(* IEC 61131-3 sources: NachHouse_CORE/V200/APP (part 15) *)

				yBtn15 := xBtn15^;

							IF j > 7 THEN
								xR^.o.ob[j].y := xR^.o.ob[7].y;			// preberie suradnicu z objektu sviatok
							ELSIF j = 7 THEN
								xR^.o.ob[j].y := xR^.o.ob[0].y - 75;			// preberie suradnicu z objektu sviatok
							ELSIF j > 0 THEN
								xR^.o.ob[j].y := xR^.o.ob[0].y;        // preberie z Pondelok
							END_IF;
							IF xO^.fn > 0 THEN								// obrazky sviatok..dovolenka
								pp	:= xR^.o.ob[j].cf.n;;                	// cislo textu
  		            	   _NhVal2(obr	:= xO^.fn + BOOL_TO_INT(xPtB^),
  		               			wO		:= xO^.w,
                              grd   := 1,
                              box   := xPtB^,                   // kruh/kruznica
                              fil   := xPtB^,                	// bude vypln
                              BgC   := xO^.FgC,						// kruznica
                              FgC   := xO^.FgC,               	// vypln
//										wL		:= 2,                      // hrubka kruznice
//									   wC    := xO^.w*20/18,              		// wl=priemer gulicky, wl=hrubka kruznice
										hB    := xO^.w*20/18,
										r		:= 10,
											);
							ELSE                                 		// dni v tyzdni, nemaju vo .fn nic
								pp	:= 201;                					// textu: den v tyzdni
  		               	_NhVal2(
                              grd   := 2,
                              crc   := true,                   // kruh/kruznica
                              fil   := xPtB^,                	// bude vypln
                              BgC   := xO^.FgC,						// kruznica
                              FgC   := xO^.FgC,               	// vypln
										wL		:= 2,                      // hrubka kruznice
									   wC    := xO^.w,              		// wl=priemer gulicky, wl=hrubka kruznice

                              txt 	:= -2,
										nTxt 	:= 21 + SINT_TO_INT(j),	// 21=PO,UT,ST
										fmt   := 2,
                              FgT   := xO^.BgC,						// farba textu
                              wT    := xO^.w/2 );
							END_IF;
							IF xR^.o.ob[0].cf.c = 1 THEN 									// vykresli objekty kopirovania
				            GC_Move  (x := 24, y := -28, GrData := xCan);
					         IF xM^.pod.cp.src = i OR (xM^.pod.cp.all AND xM^.pod.cp.dst[i]) THEN				//
					            GC_CImage   (filename := _NhFnObr(fn := 44), width := 48, height := 48,	GrData := xCan);
								ELSIF xM^.pod.cp.src = 0 THEN
									;
					         ELSIF xM^.pod.cp.dst[i] THEN
				   	         GC_CImage   (filename := _NhFnObr(fn := 38), width := 45, height := 45,	GrData := xCan);
									xM^.pod.cp.cpy := true;									// centralny prinak, ze mame nejaky ciel
								END_IF;
								IF xM^.pod.cp.all = false AND xM^.pod.cp.cpy = false THEN
									xB^.r[1].o.ob[0].wh	:= 0;
								ELSE	 //xB^.r[1].o.ob[0].cm = 130 THEN					// menu kopirovania
									xB^.r[1].o.ob[0].wh	:= 1;
									IF xM^.pod.cp.all THEN
										xB^.r[1].o.ob[0].fn := 38;						// zeleny check
										xB^.r[1].o.ob[0].cm := 132;					// browser
									ELSE
										xB^.r[1].o.ob[0].fn := 44;              	// zlte copy
										xB^.r[1].o.ob[0].cm := 130;					// copy
									END_IF;
									xB^.r[1].o.ob[0].x	:= xR^.o.ob[6].x;       // preberie znedele
									xB^.r[1].o.ob[0].y	:=	xR^.o.ob[7].y-20;			// preberie suradnicu z objektu sviatok
					         END_IF;
							END_IF;

							IF pp > 0 AND xPtB^ AND xR^.o.ob[0].set6 THEN		// vypisuje sa text dna
  		               	_NhVal2(
										xy		:= true,
										x		:= xc,
										y		:= xR^.o.ob[7].y - xR^.o.ob[7].h,
                              txt 	:= -2,
										nTxt 	:= pp,
										fmt   := 2,
                              FgT   := 3,						// farba textu
                              wT    := 28 );
							END_IF;

      				END_IF;

           106:   // ikona typ.dna na Home/zone
                  xPtD  := ADR(xO^.cf.n); 	      // adresa premennej USINT;
						xPod	:= UDINT_TO_PTR(xPtD^);
						IF xPod^.Day < 8 THEN
	               	_NhVal2(wO:=xO^.w, obr:=269);					// cisty kalendar
	               	_NhVal2(
               			y		:= xO^.w/10,
                 			txt 	:= -2,
								nTxt 	:= 21 + USINT_TO_INT(xPod^.Day-1),
                        FgT   := 3,						// farba textu
								fmt   := 2,
                        wT   := xO^.w*10/26 );
						ELSE
	               	_NhVal2(
               			wO		:= xO^.w,
               			obr	:= 275 + (3*USINT_TO_INT(xPod^.Day-8)) );
						END_IF;

           221:  // Vypist textu s hodnotou
                  // xO^.fn      :  cislo textu vypisovane od pevne od x=50
						// ak xO^.cf.c > 0
	                  // xO^.cf.c    :  cfg DEV
   	               // xO^.cf.n    :  nd DEV
                  // xO^.FgC     :  farba textu
                  // xO^.w       :  vyska textu

                  // xO^.fmt     :  textova hodnota
                  // xO^.BgC     :  farba hodnoty
                  // xO^.h       :  vyska hodnoty

                  // xO^.x       :  x-obrazka
                  // xO^.y       :  y-textu aj obrazka

                  // xO^.BgC     :  x-ova suradnica zaciatku textu

                  yTx1 := '';
                  IF xO^.fn > 0 THEN
                     _Nh_Lang(id :=  xO^.fn ,txt := ADR(yTx1));
                  ELSIF xO^.cf.c > 0 THEN
                     IF _NhxPt(c:=xO^.cf.c, n:=xO^.cf.n, x:=81) THEN
                        aTrim(wht:=1,txt:=ADR(yTx1));
                        yTx1 := CONCAT(yTx1,' ',xPt^.cf.Name);
                        yTx1 := LEFT(yTx1,25);
                     END_IF;
                  END_IF;
                  IF yTx1 <> '' THEN
                     _NhVal2(txt:=0, fmt := 0, wt:= xO^.w, FgT := xO^.FgC ,xy:=true, x:=50, y:=xO^.y );
                  END_IF;
                  yTx1 := xO^.fmt;                                          // naformatuje hodnotu do textu
                  _NhVal2(txt:=0, fmt := 2, wt:= xO^.h, FgT := xO^.BgC, xy:=true, x:=x2-90, y:=xO^.y  );

           228:   // status [2] DEV v BRW,,Quick.... vsade
		            _Nh_FRM_Read(frm:=229);                        // obrazky pre typ NH_OBR_OPV
                  xHet  := xDev;
						CASE xR^.h.cf.c OF
                    6 : c:=0;
                  ELSE  c:=1;
                  END_CASE;
						o 		:= aCfg[xR^.h.cf.c].par;
						IF xR^.h.chk   THEN													// z webu nad regulatorm sa podhodi default par
							p := xR^.h.cf.p;
						ELSIF xO^.tch  THEN
							xDev^.al.in.par := xHet^.cf.par ;
							xDev^.al.ou.par := xHet^.cf.par ;
							p	:= xDev^.al.ou.par;
						ELSE
							p	:= xDev^.al.ou.par;
						END_IF;
						IF xO^.tch THEN
							xDev^.al.in.cmd := 1;
						END_IF;
						_NhxPar (cp := o , np := p,x:=-1006);
                  pHet  	:= xPar;
                  xPvA  	:= ADR(pHet^.par.pva);
						_NH_Het_Map_Reg();
                  _Nh_Shw_ini();
                  IF xDev^.cf.typ > _Nh_TYP THEN
                     xO^.fn      := 24;
                  ELSE
                     xO^.fn      := yFrm_229.reg[c].obr1[ xReg^.Mode, xRegMod^.wht, MIN(xDev^.al.sta,3)];
                  END_IF;
                  yRn.v[0].wO    := xO^.w;
                  yRn.v[0].obr   := xO^.fn;
                  yRn.v[0].wh    := 0;
                  _Nh_Shw_Val();

           230:   // hlavny obrazok DEV podla typu.  browse
                  yRn.v[0].wO    := xO^.w;
//						xO^.fn			:=_NhObrNbr(cf:=xO^.cf.c, t:=xDev^.cf.typ);
//							_NhTypObr(cf:=xO^.cf.c, typ:=xDev^.cf.typ);
//							xO^.fn := xObrWht^.obr;

                  _Nh_Shw_ini();

//                  yRn.v[0].obr   := xO^.fn;
//                  yRn.v[0].wh 	:= INT_TO_USINT(_NhObrNbr(cf:=xO^.cf.c, t:=xDev^.cf.typ, wh:=1));

						_NhTypObr(cf:=xO^.cf.c, typ:=xDev^.cf.typ);
						xO^.fn			:= xObrWht^.obr;
	               yRn.v[0].obr   := xObrWht^.obr;
                  yRn.v[0].wh 	:= xObrWht^.wht;

						IF yRn.v[0].wh > 0 THEN
							yRn.v[0].wO := xO^.w * 20 / 24;
//							yRn.v[0].wC := xO^.w * 20 / 20;
						ELSE
	                  yRn.v[0].wO := xO^.w;
						END_IF;

                  _Nh_Shw_Val();

           231:   // status [2] DEV v BRW,,Quick.... vsade

                  _Nh_FRM_Read(frm:=231);                      // funkcia naciatania do obr, ale strukturu 230
                  _Nh_Shw_ini();
						vr				:= xDev^.al.ou.val;
						vr		:= xDev^.al.OU.val;
						IF xR^.h.chk  AND aCfg[xR^.h.cf.c].ou THEN
							{$IFDEF __NH_DALI}
							IF xR^.h.cf.c = 43 AND xF^.cf.c = 44 THEN
			      	      dlgr  := _Nh_DL_sha(gr:=1, nd := xF^.cf.n)-100;                    // cislo GRP - 100
								xDLs 	:= xDEv;
								vr 	:= USINT_TO_REAL(xDLs^.cx.scn.lvl[dlgr]);
							ELSIF xR^.h.cf.c = 44 AND xF^.cf.c = 43 THEN
								dlgr  := _Nh_DL_sha(gr:=1, nd := xR^.h.cf.n)-100;                    // cislo GRP - 100
								_NhxPt(c:=xF^.cf.c, n:=xF^.cf.n,x:=-135);
								xDLs 	:= xPt;
								vr 	:= USINT_TO_REAL(xDLs^.cx.scn.lvl[dlgr]);
							ELSIF aCfg[xO^.cf.c].par > 0 THEN
							{$ELSE}
							IF aCfg[xO^.cf.c].par > 0 THEN
							{$END_IF}

                   		IF _NhxPar(cp := aCfg[xO^.cf.c].par, np := xR^.h.cf.p ,x:=238) THEN
									vr		:= USINT_TO_REAL(xPar^.all.lvl);
								ELSE
									;
//									vr		:= xDev^.al.ou.val);
								END_IF;
							END_IF;
							IF vr > 0.0  THEN
								yRn.v[0].txt 	:= 3;													// vypise sa to co je vo vr
								yRn.v[0].wh    := 21;												// pri check, je vzdy zeleny podklad
							ELSE
								yRn.v[0].wh  := 10;													// sivy podklad OFF
							END_IF;
						ELSE
	      				s 				:= xDev^.al.sta;
							IF s > 0 THEN
								s	:= 2;
							ELSE
								s	:= 0;
							END_IF;
							IF  yFrm_231.dev[xO^.cf.c,s] < 0 THEN
								p := yFrm_231.dev[xO^.cf.c,2] * -1  + USINT_TO_INT(xDev^.al.sta-1);
								p	:= MIN(p,50);						// opravit
								IF yFrm_231.sta[p, 0] < 0 THEN
		      	            yRn.v[0].txt   := INT_TO_SINT( yFrm_231.sta[p, 0] * -1 );
		         	         yRn.v[0].obr   := 0;
								ELSE
		               	   yRn.v[0].obr   := yFrm_231.sta[p, 0];
								END_IF;
  			               yRn.v[0].wh    := INT_TO_USINT(yFrm_231.sta[p, 1]);
(*
							ELSIF xO^.cf.c = 4 	AND vr < 100.0 THEN						// SCN nie je naplno
	         	         yRn.v[0].obr   := 0;
								IF vr  > 0.0 THEN
			         	      yRn.v[0].wh    := 11;
								ELSE
			         	      yRn.v[0].wh    := 10;
								END_IF;
*)
							ELSIF xO^.cf.c = 4  THEN						// SCN nie je naplno
								yRn.v[0].obr   := 207;
								IF vr >= 100.0 THEN
			         	      yRn.v[0].wh    := 14;
								ELSIF vr  > 0.0 THEN
			         	      yRn.v[0].wh    := 17;
								ELSE
									yRn.v[0].obr   := 0;
									yRn.v[0].wh    := 10;
								END_IF;

							ELSIF xO^.cf.c = 44 	AND vr < 100.0 THEN            			// DLg scen nie je naplno
	         	         yRn.v[0].obr   := 0;
								IF vr  > 0.0 THEN
			         	      yRn.v[0].wh    := 11;
								ELSE
			         	      yRn.v[0].wh    := 10;
								END_IF;
							ELSE
	         	         yRn.v[0].obr   := yFrm_231.dev[xO^.cf.c,s];
   	         	      yRn.v[0].wh    := INT_TO_USINT(yFrm_231.dev[xO^.cf.c,s+1]);
							END_IF;
						END_IF;

(*
						IF xO^.cf.c = 44 THEN														// DLg nema Check
							IF xDev^.al.ou.val >=254 THEN
								yRn.v[0].wh  := 102;													// Oranzovy ON = kompletne zapnuta scena
							END_IF;
                  ELSIF aCfg[xO^.cf.c].ou AND xR^.h.chk AND aCfg[xO^.cf.c].par > 0  THEN   // pre OUT-DEV vp vazbe
     						yRn.v[0].obr	:= 0;                                     // zrusi obrazok, aby sa nezmensoval podklad
							yRn.v[0].FgT   := 1;													// pri check, je vzdy zeleny podklad
							IF xF^.cf.c = 44 THEN
								yRn.v[0].wh    := 13;												// pri check, je vzdy zeleny podklad
								{$IFDEF __NH_DALI}
	 							dlgr	:= _Nh_DL_sha(gr:=1,nd := xF^.cf.n)-100 ;				// 0..15
								xDLg	:= xDev;
								vr		:= MIN(100,USINT_TO_REAL(xDLs^.cx.scn.LVL[ dlgr ]));
								IF vr > 0.0 THEN
									yRn.v[0].txt := 3;													// vypise sa to co je vo vr
								ELSE
									yRn.v[0].wh  := 10;													// sivy podklad OFF
								END_IF;
								{$END_IF}

                     ELSIF _NhxPar(cp := aCfg[xO^.cf.c].par, np := xR^.h.cf.p ,x:=238) THEN
								yRn.v[0].wh    := 13;												// pri check, je vzdy zeleny podklad
								vr	:= MIN(100,USINT_TO_REAL(xPar^.all.lvl));
								IF aCfg[xO^.cf.c].analog THEN
									yRn.v[0].txt := 3;													// vypise sa to co je vo vr
								ELSIF vr > 0.0 THEN
									yRn.v[0].txt := 2;													// vypise sa to co je vo vr
								ELSE
									yRn.v[0].wh  := 10;													// sivy podklad OFF
								END_IF
							END_IF;
                  END_IF;
*)
					   IF yRn.v[0].wh > 0 AND yRn.v[0].obr > 0 THEN								// obrazok ma podklad, zmensi sa
	                  yRn.v[0].wO := xO^.w*20/23;
					   END_IF;

                  _Nh_Shw_Val();

           232:   // HOME-DASH, Cat/hlavny obr + CAT/status
                  _Nh_FRM_Read(frm:=232);                      // funkcia naciatania do obr, ale strukturu 230
                  p := xO^.cf.n;                                                      // cislo CAT
						_NhxRoW(nbr := xA^.sbj, zon := true);
						_NhxZon(c:=3, nz:=xA^.sbj, x:=111);
						IF xRoW^.cat[p] THEN																// hlavna ikona   je j=1
							c := 1;
						ELSE
							c := 0;
						END_IF;

					   CASE p OF
                    6 : // PSN
								c := xZon^.cx.lck.stat;
								IF xZon^.cx.lck.stat > 9 THEN
									c := 2;
								ELSIF c = 2 AND xZon^.cx.lck.AllLocked = false THEN
									c := 10;
								END_IF;
		                  IF xL^.obj = 0 THEN
    								x4o   := ADR(xB^.r[4].o.ob[p]);
									x4o^	:= yFrm_232.psn4;
									ok		:= 0;
									IF xHoW^.BodyOu THEN
										x4o^.ok[1]  := 1;
										ok				:= 0;
									END_IF;
									IF xHoW^.BodyIn THEN
										x4o^.ok[2]  := 1;
										ok				:= 0;
									END_IF;
									_Nh_Shw_LCK_ET(sta:=xZon^.cx.lck.stat, et:=xZon^.cx.lck.et, o := 4);
									IF ok THEN
//										x4o^.wh	:= 0;
									END_IF
								END_IF;

                  ELSE
                  ;
                  END_CASE;
				  		_Nh_Shw_ini();
						_Nh_Shw_232(o1 := xL^.obj > 0 AND j=1,  cat := p, sta := c);     	// pre j=1 hlavna ikona sa je iny obrazok
                  _Nh_Shw_Val();

           233:   // OBR Quick menu

                  _Nh_FRM_Read(frm:=233);                      // funkcia naciatania do obr, ale strukturu 230
                  _Nh_Shw_ini();
                  yRn.v[0].wO    := xO^.w;
                  yRn.v[0].obr   := yFrm_233.dev[xO^.cf.c].obr[xDev^.al.sta];
                  yRn.v[0].wh    := yFrm_233.dev[xO^.cf.c].wht[xDev^.al.sta];
                  IF yRn.v[0].wh > 0 THEN
                     yRn.v[0].wC   := 80;
                     yRn.v[0].wO   := 64;
                  ELSE
                     yRn.v[0].wO   := 80;
                  END_IF;
                     yRn.v[1].ok    := true;
                     yRn.v[1].txt   := 101;
                     yRn.v[1].wT    := 16;
//                     yRn.v[1].fmt   := 2;
                     yRn.v[1].y     := 55;   //xO^.w*10/13;

//                     xO^.w    := 64;

                  CASE xO^.cf.c OF
//                      1 :  ;// ZAS
                     222 :  ;// ZAS
//                      21 :  ;// ZAS
//                      37 :  ;// GAR/BRA
//                      42 :  ;// DLS
                  ELSE
                  ;
                  END_CASE;

                  _Nh_Shw_Val();

           234:   // ROM/ZON/PSN + teplota/status
				      _Nh_FRM_Read(frm:=231);                      // funkcia naciatania do obr, ale strukturu 230
                  _Nh_Shw_ini();
						IF xL^.obj = 50  THEN												// ZON->ACT
							CASE j OF
                       1 : // hlavny obr
									yRn.v[0].obr   := 69;	//yFrm_231.sta[2, 0];
   		               	yRn.v[0].wh    := 0;
                       6 : // stavovy obr
           						i := 0;
									IF xR^.h.chk AND xR^.h.nd > 0 THEN
										_NhxVaz(cv:=xL^.vaz, nd := xR^.h.nd);
										IF _NhxPar(cp := aCfg[3].par, np:= xVaz^.in.p ,x:=239) THEN
											pZon 	:= xPar;

										IF  pZon^.cmd < 60 THEN
											pZon^.cmd := 60;
										ELSIF pZon^.cmd > 69 THEN
											pZon^.cmd := 60;
										END_IF;

											i 		:=	pZon^.cmd - 60 ;
										END_IF;
										yRn.v[0].obr   := yFrm_231.sta[i, 0];
        								yRn.v[0].wh    := INT_TO_USINT(yFrm_231.sta[i, 1]);
                  			ELSE
										yRn.v[0].obr   := yFrm_231.sta[i, 0];
   			               	yRn.v[0].wh    := INT_TO_USINT(yFrm_231.sta[i, 1]);
									END_IF;
							END_CASE;
						ELSIF xL^.psn  THEN
							xRom	:= xDev;
				         xLck  := ADR(xRom^.cx.lck);
							p		:= yFrm_231.dev[xR^.h.cf.c,2];
							c		:= xLck^.stat;
							IF xLck^.stat > 9 THEN
								c := 2;
							END_IF;
							IF c > 0 AND  p < 0 THEN
													//	1.riadok                         // 1.riadok je stat:=1
								p 					:= yFrm_231.dev[xR^.h.cf.c,2] * -1  + USINT_TO_INT(c-1);
								IF xR^.h.cf.c = 3 AND p = 2 AND xLck^.AllLocked = false THEN
									p := 10;
								END_IF;
		                  yRn.v[0].obr   := yFrm_231.sta[p, 0];
   		               yRn.v[0].wh    := INT_TO_USINT(yFrm_231.sta[p, 1]);
							ELSE
								s 					:= c * 2;														// 0: [0..1] 1: [2..3]
		                  yRn.v[0].obr   := yFrm_231.dev[xR^.h.cf.c,s];
   		               yRn.v[0].wh    := INT_TO_USINT(yFrm_231.dev[xR^.h.cf.c,s+1]);
                     END_IF;

	                  yRn.v[0].wC 	:= xO^.w;
	                  yRn.v[0].wO 	:= xO^.w*20/24;
						ELSE
	                  yRn.v[0].obr   := 0;
   	               yRn.v[0].wh    := 100;
						END_IF;
                  _Nh_Shw_Val();

           240:   // obrazky nad DSH + domcek
                  p := xO^.w - 10;
                  CASE xO^.cf.p OF                                               // cislo CAT
                    1 : ii := 0; p := xO^.w;                                     // Domcek
                    2 : ii := 0; p := xO^.w;                                     // sviecka vnutri
                    3 : ii := 0; p := xO^.w;                                     // Okno
                    4 : ii := 0; p := xO^.w;                                     // Fotovoltaika
                    5 : ii :=22;                                                 // Dvere - oranzova
                   10 : ii := 0; p := xO^.w;                                     // Dvere - oranzova
                  ELSE
                     ii    := 23;
                  END_CASE;
                  _NhVal2( wh := ii, obr := xO^.fn, wO := p);
                  IF xO^.tch  THEN
                     xO^.tch := false;
                  END_IF;

           255:   // riadok prihlaseneho usra na webserveri
                  xR^.h.cf.n := MIN(xR^.h.cf.n,7);

                  CASE aAcc.wa[xR^.h.cf.n].state OF
                     SESSION_EMPTY  : yTx1 := 'EMPTY ';
                     SESSION_LOGIN  : yTx1 := 'LOGIN ';
                     SESSION_ACTIVE : yTx1 := 'ACTIVE';
                     SESSION_LOGOUT : yTx1 := 'LOGOUT';
                  ELSE                yTx1 := '??????';
                  END_CASE;
                  yTx2  := IPADR_TO_STRING(IPAdr := aAcc.wa[ xR^.h.cf.n ].IP );
                  aBlank(txt := ADR(yTx2), n:= 18);
                  yTx3 := LEFT(targetPage,10);
                  yTx1  := CONCAT(INT_TO_STRING(xR^.h.cf.n),'  ', yTx1,'    ',yTx2,'  ', yTx3); //111,'%d');
                  _NhVal2(   txt:=0, wT:=22, FgT:=4, fmt:=0);
                  yTx1  := LEFT(aAcc.wa[ xR^.h.cf.n ].LastFile,30);
                  _NhVal2(   txt:=0, wT:=22, FgT:=3, fmt:=0, y := 40);
         END_CASE;
      END_IF;
      j := j + 1;
   END_WHILE;
END_FUNCTION

{ $ END_IF }

(* ---- _Nh_IMP_CFG.st ---- *)
(* IMPORT from NH2.exp *)

VAR_GLOBAL
	xHw      	{HIDDEN} 	: PTR_TO NH_DEV_HW5;
	yFrm_500	AT mObr			{HIDDEN} : NH_FRM_500;					// import from NH2.exp
	yFrm_250	AT mObr			{HIDDEN} : NH_FRM_250;					// import from NH2.exp
	yImp		AT yFrmData		{HIDDEN} : NH_LOG_IMP;					// only struct import
END_VAR

FUNCTION _Nh_Import_CIB_Find_ID {HIDDEN}   : BOOL
	VAR_INPUT
		ok		: BOOL;
		cf		: USINT;
		ID		: STRING[5];
	END_VAR
	nDel	:= 0;
	_Nh_Import_CIB_Find_ID := false;
   FOR nd := 1  TO aCfg[cf].rec DO
      IF _NhxPt(c:=cf, n:=nd, ok:=ok, x:=3) THEN
	      IF xPt^.ok.ok AND xPt^.cf.ID = ID THEN
				_Nh_Import_CIB_Find_ID := true;
				EXIT;
			ELSIF nDel > 0 THEN
				;
   	   ELSIF xPt^.ok.ok=false AND xPt^.cf.ID = '' THEN
				_Nh_Import_CIB_Find_ID := true;
				nDel 	:= nd;
				xDel	:= xPt;
	      END_IF;
		END_IF;
   END_FOR;
END_FUNCTION

FUNCTION _Nh_Import_CIB_To_MEM {HIDDEN}   : BOOL
	_Nh_Import_CIB_To_MEM := true;
	WHILE true DO
		cf	:= STRING_TO_USINT(yImp.cf);
		IF _Nh_Import_CIB_Find_ID(ok:=true, cf:=cf, ID:=yImp.ID) THEN
			IF nDel > 0 THEN
				xPt	:= xDel;
				nd		:= nDel;
				y:=y+1;
			ELSE
				x:=x+1;
			END_IF;
			xDev	:= xPt;

			xDev^.ok.ok		:= true;
			xDev^.cf.ID		:= yImp.ID;
			xDev^.cf.idx 	:= nd;
			yImp.NameCf		:= xDev^.cf.Name;
			IF yImp.Name = '' THEN
				;
			ELSIF xDev^.cf.Name = '' THEN
				xDev^.cf.Name := yImp.Name;
			END_IF;

			IF yImp.cfg <> 'ROM' THEN
				IF yImp.cfg = 'TLA'  THEN
					xDev^.cf.typ := MAX(xDev^.cf.typ,STRING_TO_SINT(yImp.Typ));
//			 	ELSIF aSys.NewDBX THEN
			 	ELSIF yImp.typYes = 'Y' THEN
					xDev^.cf.typ := STRING_TO_SINT(yImp.Typ);
				END_IF;
			 	IF aSys.NewDBX THEN
	            xDev^.cf.Inv :=  STRING_TO_BOOL(yImp.inv);
				END_IF;
           	// aktualizuju sa HW adresy
				xHw   := xDev + 1 + USINT_TO_UDINT( aCfg[cf].cf) + USINT_TO_UDINT(aCfg[cf].al) + aCfg[cf].cx;
            i     := STRING_TO_USINT(yImp.d) ;                           // pocet HW-adries  1=0, lebo sa zadina d.[0]
            xHw^.typ :=  STRING_TO_USINT(yImp.HWtyp);
//            xHw^.cfg :=  yEx1.hw.cfg;

			 	xHw^.d[i] := STRING_TO_UDINT(yImp.HWs);
				IF  yImp.RomID <> '' THEN
					IF _Nh_Import_CIB_Find_ID(cf:=1,ID:=yImp.RomID) THEN
						yImp.rom		:= INT_TO_STRINGF(nd,'%3u');
						IF xDev^.cf.rom = 0 THEN
							xDev^.cf.rom := INT_TO_USINT(nd);
						END_IF;
					END_IF;
         	END_IF;
			ELSE	// ROM,ZON
				IF xDev^.cf.rom = 0 THEN       		// rom,zone
					xDev^.cf.rom := STRING_TO_USINT(yImp.rom);				// nadradena zona
				END_IF;
				IF aSys.NewDBX THEN
					xDev^.cf.typ := STRING_TO_SINT(yImp.TypRom);
				END_IF;
			END_IF;
			EXIT;
		ELSE
			z:=z+1;
			aCfg[cf].new := aCfg[cf].new + 1;
			_Nh_Go_DbxToMem(ForceRamOk:=true);
		END_IF;
	END_WHILE;
	yImp.ok := '1';
	fbLine(write:=true,seek:=fbLine.LineS);
END_FUNCTION

FUNCTION_BLOCK _Nh_Import_CIB	// kopia vsetkych, alebo modifikovanych CFG/PAR/VAZ na USB (z MEM/RAM/DBX)
	VAR_INPUT
		Go				: USINT;
	END_VAR
	VAR_OUTPUT
		Done			: BOOL;
		busy			: BOOL;
		err			: BOOL;
//		nExp			: UINT;
//		cyc			: UINT ;
	END_VAR
	VAR

	END_VAR
	done	:= false;
	CASE Go OF
     	0:	RETURN;
     	1:		// start import
				x	:= 0;
				_Nh_FRM_Read(frm:=500);
				yTx2	:= CONCAT('.Import from: ',_Nh_EXP);
				_Nh1RowTxt(logRst:=1);
				yTx1		:=  _Nh_EXP;
           	fbFileRWa(init:=true,exec:=true,line:=true, adrVar:=PTR_TO_UDINT(ADR(yTx0)),fileName:=yTx1);
				IF fbFileRWa.errID > 0 THEN
					Go	:= 99;
				ELSE
					busy	:= true;	grp:=0;
					Go		:= 11;
					_Nh_Log_Path(wh:=22, frm:=1, wh2:=1);
//					yTx0	:= CONCAT(yTx1, DT_TO_STRINGF(aSys.NhDT,'%TDD_hhmm.cib') );
					yTx0	:= yTx1;
					yTx2	:= CONCAT('.Import to: ',yTx0);
					_Nh1RowTxt(logRst:=1);
					fbLine(open:=true,del:=true,seek:=0,nLine:=1, aLine:=PTR_TO_UDINT(ADR(yImp)) ,sLine:=SIZEOF(yImp));
				END_IF;

		16:	// prejde DEV ine ako ROM a podla RomID zisti cislo ROM
				IF fbLine.LineS = 0 THEN
					grp:=0;x:=0;y:=0;z:=0;
					yTx2 	:= '..Start check Dev' ;
					_Nh1RowTxt(logRst:=1);
				END_IF;
				grp:=grp+1;          											// pocitadlo cyklov
				WHILE go=16 DO	// _NhMaxRWLimit() //OR _NhMaxTimeCyc()
					fbLine(write:=false,seek:=fbLine.LineS+1);
					IF fbLine.done AND yImp.cfg <> 'ROM' THEN

						_Nh_Import_CIB_To_MEM();

//						yTx2	:= CONCAT('...Dev: ',yImp.CFG,'  ',TIME_TO_STRINGF(SUB_DT_DT(GetRtc(),aSys.NhDT),'%Ts.zzz'),'  ',UDINT_TO_STRING(aSys.RWtoFileCycle) );
//						_Nh1RowTxt(logRst:=1);
						IF _NhMaxRWLimit() OR _NhMaxTimeCyc() THEN
							EXIT;
						END_IF;
					END_IF;
					IF fbLine.LineS = 0 THEN
						yTx2	:= CONCAT(	'..End   check Dev.',	TIME_TO_STRINGF(_NhGetTimeCyc(),' %Ts.zzz '),
												'cyc',INT_TO_STRINGF(grp,'%3u ' ),
												'x:',	INT_TO_STRINGF(x,'%4u '),
												'y:',	INT_TO_STRINGF(y,'%4u '),
												'z:',	INT_TO_STRINGF(y,'%4u '),
												'rw:',  UDINT_TO_STRINGF(aSys.RWtoFileCycle,' %7u ' )
											);
						_Nh1RowTxt(logRst:=1);
//						Go	:= 19;
						Go	:= 99;
					END_IF;
				END_WHILE;

		15:	// prejde ROM a podla RomID zapise cislo vety do ROM
				IF fbLine.LineS = 0 THEN
					grp:=0;x:=0;y:=0;z:=0;
					yTx2 	:= '..Start check ROM' ;
					_Nh1RowTxt(logRst:=1);
				END_IF;
				grp:=grp+1;
				WHILE go=15 DO
					fbLine(write:=false,seek:=fbLine.LineS+1);
					IF fbLine.done AND yImp.cfg = 'ROM' THEN
						_Nh_Import_CIB_To_MEM();

						IF _NhMaxRWLimit() OR _NhMaxTimeCyc() THEN
							EXIT;
						END_IF;
					END_IF;
					IF fbLine.LineS = 0 THEN
						yTx2	:= CONCAT(	'..End   check ROM.',TIME_TO_STRINGF(_NhGetTimeCyc(),' %Ts.zzz '),
												'cyc',INT_TO_STRINGF(grp,'%3u ' ),
												'x:',	INT_TO_STRINGF(x,'%4u '),
												'y:',	INT_TO_STRINGF(y,'%4u '),
												'z:',	INT_TO_STRINGF(y,'%4u '),
												'rw:',  UDINT_TO_STRINGF(aSys.RWtoFileCycle,' %7u ' )
											);
						_Nh1RowTxt(logRst:=1);
						Go	:= 16;
					END_IF;
				END_WHILE;

		19:	//

            { $IFDEF __NH_WRK }
               _NhDataWrk();
            { $END_IF }

		11:	// prejede /NH2.exp, vytvori z neho /RAM/EXP/cib.CSV
//				yTx1		:=  _Nh_EXP;
				grp:=grp+1;          											// pocitadlo cyklov
				WHILE Go=11 DO
					fbFileRWa(fileName:=yTx1);
					IF fbFileRWa.done OR fbFileRWa.errID > 0	THEN
						yTx2	:= CONCAT('.End Import.',TIME_TO_STRINGF(_NhGetTimeCyc(),' %Ts.zzz '),
													 'cyc:',  INT_TO_STRINGF(grp,'%5u '),
													 'rec:',  INT_TO_STRINGF(x,'%5u ' ),
													 'rw:',  UDINT_TO_STRINGF(aSys.RWtoFileCycle,' %7u ' )
											);
						_Nh1RowTxt(logRst:=1);
						fbLine.LineS:=0;
						Go := 15;
					ELSIF fbFileRWa.row THEN
						j := FIND(yTx0,' AT %');
            		IF j > 0 THEN                                                     // len veta, ktora ma adresu
//							yTx2 	:= CONCAT(UDINT_TO_STRINGF(aSys.RWtoFileCycle,'%10u '), TIME_TO_STRING(SUB_DT_DT(GetRtc(),aSys.NhDT)),'  ',yTx0) ;
//							_Nh1RowTxt(logRst:=1);
							x			:= x + 1;
							yImp		:=  yFrm_500.eImp;
							yImp.cfg	:= MID(yTx0,3,1);
               		cf    	:= _NhGetCFG(cfg := yImp.cfg);                               // zisti ci mame taketo dev
							yImp.cf	:= USINT_TO_STRINGF(cf,'%3u');
							ok    := false;
               		IF cf = 0 THEN                                                // nezname CFG
								yTx2 	:= CONCAT('...Unknown cfg: ',yTx0) ;
								_Nh1RowTxt(logRst:=1);
               		ELSIF acfg[cf].imp THEN                      				// toto DEV sa importuje
								yImp.ID	:= MID(yTx0,3,5);   STRING_TO_UPPER(yImp.ID);
								yTx3					:= MID(yTx0,5,8);   STRING_TO_UPPER(yTx3);
		                  IF yTx3 = ' AT %' THEN                                 // nema priponu
//                     		yImp.TYP   := ' ';
                 			ELSE
                     		yImp.TYP   := MID(yTx3,1,2);
                  		END_IF;
                  		IF yImp.ID <> 'ROM' THEN                                   // ROM nema adresu
		                     // podla typu premennej sa ulozi zdresa oblasi
      		               IF 	FIND(yTx0,'%QB') > 0 THEN        // vystup
                              yImp.IO   := 'Q';
	                           {asm}
   	                           LEA %Y0
      	                        WR  Base0
         	   	  	         {end_asm}
            		         ELSIF 	FIND(yTx0,'%IB') > 0 THEN        // vstup
                           	yImp.IO   := 'I';
                           	{asm}
          	                  	LEA %X0
	                              WR  Base0
   	                        {end_asm}
      		               ELSIF 	FIND(yTx0,'%MB') > 0 THEN        // pamat
            	               yImp.IO   := 'M';
                           	{asm}
	                        	  LEA %R0
   	                     	  WR  Base0
      	                     {end_asm}
									END_IF;
         	            END_IF;
	                     j     := FIND(yTx0,'AT %');                       // 'WSB_101_4 AT %IB486.0 : BOOL;
	                     yTx0  := DELETE(yTx0,j+5,1);                      // '486.0 : BOOL;
	                     j     := FIND(yTx0,' : ');
	                     yTx3  := MID(yTx0,j-1,1);                         // '486.0'
	                     j     := FIND(yTx3,'.');
	                     IF j > 0 THEN                                      // yTx3    '172.3'
                           yImp.MEM   := 'B';
                           _LangTXT   := MID(yTx3,j-1,1);                    // '172'
                           yTx3  := DELETE(yTx3,j,1);                   // '3 :'
                           sz    := (Base0 + STRING_TO_UDINT( _LangTXT ) ) * 8 + STRING_TO_UDINT( yTx3 );
   	                  ELSE
                           yImp.MEM   := 'R';
                           sz := Base0 + STRING_TO_UDINT(yTx3);         // '172'
      	               END_IF;
//         	            yImp.HW   := sz;
         	            yImp.HWs  := UDINT_TO_STRINGF(sz,'%8u');

	                  	// nazov, miestnost
		                  j := FIND(yTx0,'(*');                     // zaciatok poznamky
   		               IF j > 0 THEN
      		               yTx0  := DELETE(yTx0,j+2,1);           // odreze zaciatok a zostane : ' nazov DEV ; rom ; nazov miestnosti
         		            j     := FIND(yTx0,'*)');					// koniec poznamky
               	      	yTx0  := DELETE(yTx0,3,j-1);           // odreze koniec
	               	      j := FIND(yTx0,';');                   // za nazvom je cislo miestnosti			'nazov;104'
	                  	   IF j > 0 THEN
   	                  	   yImp.Name 	:= MID(yTx0,j-1,1);      	// zapise nazov         		'nazov'
	                        	yTx0        			:= DELETE(yTx0,j,1);    	// odreze zaciatok 				'104' .. ' 104'
		                     	aTrim(txt := ADR(yTx0), wht := 1);        		// zo vsetkych stran odstrani medzewry
      	                  	IF yImp.cfg = 'ROM' OR yImp.cfg = 'ZON' THEN
											yImp.TypRom	:= yTx0;  					// pripadny typ ROM -1=nezaradene
            	               	yImp.RomID  := yImp.ID;    // co zostalo je ROM
               	         	ELSE
                  	         	yImp.RomID  := yTx0;              // co zostalo je ROM
										END_IF;
							      END_IF;
            	        		aTrim(txt := ADR(yImp.Name), wht := 1);        // zo vsetkych stran odstrani medzewry
   	                  ELSE
      	                  yImp.Name  := '';
         	            END_IF;     // koniec hladania nazvu

//                        yImp.typYes	:= ' ';

				            j  := STRING_TO_SINT(yImp.TypRom);
								i	:= 1;
					         IF cf = 1 THEN
									CASE j OF
                             1 : i := 3;					// vnutorna miestnost -> 1.NP
                             2 : i := 2;					// vonkajsia miestnost -> Vonku
                             3 : i := 5;              // podzemna  miestnost -> Podzemie
									ELSE i := 1; 					// ostatne -> domcek
                           END_CASE;
									yImp.Rom 	:= USINT_TO_STRINGF(i,'%3u');
									yImp.TypRom :=  SINT_TO_STRINGF(j,'%1d');
					         ELSIF cf = 3 THEN
									CASE j OF
                             2 : i := 2;					// vonkajsia zona -> Vonku
									ELSE 	i := 1; 					// ostatne -> domcek
                           END_CASE;
									yImp.Rom 	:= USINT_TO_STRINGF(i,'%3u');
									yImp.TypRom :=  SINT_TO_STRINGF(j,'%1d');
				         	ELSIF yImp.typ   = 'Q' THEN                    // vystup d[0]
					            yImp.d := '1';
					         ELSIF yImp.typ   = 'Y' THEN                    // vystup d[2]
					            yImp.d := '2';
					         ELSIF yImp.typ   = 'R' THEN
					            ;
					         ELSIF yImp.typ   = 'G' THEN
					            yImp.d  := '1';
					         ELSIF yImp.typ   = 'B' THEN
						         yImp.d := '2';
					         ELSIF yImp.typ   = 'W' THEN                    // WW
						         yImp.d := '3';
					         ELSIF yImp.typ   = 'C' THEN                    // CW
						       	yImp.d := '5';
					         ELSIF yImp.typ   = 'U' THEN                    // ROL-up
               				;
					         ELSIF yImp.typ   = 'D' THEN                    // ROL-Dn
					            yImp.d  := '1';
					         ELSIF yImp.cfg   = 'TLA' THEN                  // tlacitko bude mat typ najvacsi
                        	yImp.typYes	:= 'Y';
	            	         IF yImp.typ = '0' OR yImp.typ = ' ' THEN                                                      // zapni = vypni (inverzia),
										yImp.typ := '1';
									END_IF;
                           i := STRING_TO_USINT(yImp.typ)- 1;
						       	yImp.d := USINT_TO_STRINGF(i,'%1u');
					         ELSE  ok := true;
                        	yImp.typYes	:= 'Y';
				               CASE cf OF
				                   21 :    // ZAS
				            	         IF yImp.typ = '1' THEN                                                      // zapni = vypni (inverzia),
				         	               yImp.inv := '1';
													ok				 := false;		                                     // nema vplyv na typ, urcuje sa v SW
				   	                  END_IF;
				                   15 :    // PIR
				            	         IF yImp.typ = '0' THEN                                                      // zapni = vypni (inverzia),
				         	               yImp.inv := '1';
				   	                  END_IF;
				                    8 : ;  //TVE
				                   23 : ;  //REK
            			      END_CASE;
					         END_IF;

//					         IF i < 255 THEN
									IF yImp.MEM = 'R' THEN														// z exportu sa samo oznaci podla typu premennej R/B
						            yImp.HwTyp := '1';                                				// 0=bool,1=real
									END_IF;
//					          	xExp^.hw.d[i] := xRwa^.hw;                                		// HW adresy
//					         END_IF;

								fbLine(append:=true);
							ELSE
								yTx2 	:= CONCAT('..No imported: ',yTx0) ;
								_Nh1RowTxt(logRst:=1);
							END_IF;

						END_IF;
					END_IF;
					IF _NhMaxRWLimit() OR _NhMaxTimeCyc() THEN
//   					EXIT;
					END_IF;
				END_WHILE;

//				aSys.ini := 217;
//				RETURN;

		99:	//
				fbLine(close:=true,seek:=0);
				done	:= true;
				busy	:= false;
				Go		:= 0;
	END_CASE;
END_FUNCTION_BLOCK

(* ---- prgMain.ST ---- *)
{ $ IFNDEF _Nh_CUST_RESTART } 	                 // ak nie je definovana funkcia v uzivatelskom subore, vytvori sa pre
(*
   FUNCTION _Nh_CUST_RESTART  {HIDDEN} : BOOL
		;
   END_FUNCTION
*)
{ $ END_IF }

TYPE _Nh_Last_State_ON : STRUCT 		// last state PRG/CPU before restart
		lastDT:		DT; (* Comment *)
		Ini: 			USINT;
		copy:		BOOL;
		cfg:		BOOL;

	END_STRUCT
END_TYPE

VAR_GLOBAL
//DeleteFiles : DeleteSurplusFilesEx := ( delEmptyDir := true ); // delete surplus files in  given  directory
  	fb_Nh_Import_CIB		: _Nh_Import_CIB;
	fb_Nh_Cfg_Restart		: _Nh_Cfg_Restart;
	fb_Nh_Log_DBX_RW		: _Nh_Log_DBX_RW;		// write log to buffer (DBx,RBx) and read from buffer and send datagram to Pi or Write to USB/LOG
END_VAR
VAR_GLOBAL RETAIN
	_NhLastPowerOffState		: _Nh_Last_State_ON; 		// last state PRG/CPU before Power OFF
END_VAR

PROGRAM prgMain
   VAR
   	fbCrHet				: _Nh_Create_HET;
      { $ IFDEF __NH_WEB }
         fbWebControl   : _NhWebControl;
      { $ END_IF  }
		ok				: BOOL;
//    	notification 	: TWebPushNotif;
//    	webPush      	: fbWebPushService;

   END_VAR
//	rb 							:= 1;
	aSys.RWtoFileCycle		:= 0;																	// how many writes to all files in cyc
	aSys.NhTime    			:= GetTime();
  	aSys.NhDate    			:= GetDate();
  	aSys.NhDT      			:= GetDateTime();													// skoro strojovy cas zaciatku cyklu, ked sa uz zapli vsetky vystupy
  	aSys.LogHed.logTime  	:= TIME_TO_STRINGF(aSys.NhTime,'%Thh:mm:ss.zz');
  	aSys.LogHed.logDate  	:= DATE_TO_STRINGF(aSys.NhDate,'%TYY-MM-DD');

	// 1   SEC 	=  10000 SYSTEM_S.LAST_CYCLE_TIME_100US      1.0 * 10 000
	// 0,7 SEC 	=  7000 SYSTEM_S.LAST_CYCLE_TIME_100US	   	0.7 * 10 000
	// 0.001    =    10
   aSys.dMin      	:= USINT_TO_INT( SYSTEM_S.COUNTER_HOURS ) * 60 + USINT_TO_INT(SYSTEM_S.COUNTER_MINUTES);  // pocet minut v ramci dna
	aSys.rSec	   	:= UINT_TO_REAL( SYSTEM_S.LAST_CYCLE_TIME_100US ) / 10.0 ;		// REAL: doba minuleho cyklu v mS (prevod zo 100 mikrosekund)
	aSys.mSec			:= REAL_TO_UINT( ROUND(  aSys.rSec ) );			            // UINT: doba minuleho cyklu v mS  (prevod zo 100 mikrosekund)
//	aSys.rTime     	:= TIME_TO_REAL(aSys.NhTime);				// REAL: cas v sekundach od polnoci

(*
	IF System_S.F_EDGE_10SEC THEN	//System_S.F_EDGE_1MIN OR  System_S.R_EDGE_1MIN THEN				// kazdych 30sec
		aSys.LogHed.Quite10Sec := aSys.LogHed.Quite10Sec + 1;
		IF aSys.LogHed.Quite10Sec > 6 THEN														// ak nebol 1 min zapis, zavrie subor
			rb := _Nh_Log_Evn_ADD(tsk := 255);
		END_IF;
		aSys.mSecMax			:= 0;
	END_IF;
*)

 	aSys.mSecMax 	:= MAX(aSys.mSec, aSys.mSecMax);
	aSys.et50		:= aSys.et50 + SYSTEM_S.LAST_CYCLE_TIME_100US;
	IF aSys.PULSE_BEEP THEN
		IF aSys.et_PULSE_BEEP > aSys.mSec THEN
			aSys.et_PULSE_BEEP := aSys.et_PULSE_BEEP - aSys.mSec;
		ELSE
			aSys.PULSE_BEEP 		:= 0;
			aSys.et_PULSE_BEEP 	:= 1000;
		END_IF;
	ELSIF asys.et_PULSE_BEEP > aSys.mSec THEN
		aSys.et_PULSE_BEEP := aSys.et_PULSE_BEEP - aSys.mSec;
	ELSE
		aSys.PULSE_BEEP		:= 1;
		aSys.et_PULSE_BEEP	:= 200;
	END_IF;

	IF aSys.et50 >= 500 THEN
		aSys.et50			:= 0;
		aSys.u50ms			:= 1;
		aSys.PULSE_50MS 	:= NOT aSys.PULSE_50MS;
	ELSE
		aSys.u50ms			:= 0;
	END_IF;
	aSys.et100		:= aSys.et100 + SYSTEM_S.LAST_CYCLE_TIME_100US;
	IF aSys.et100 >= 1000 THEN
		aSys.et100			:= 0;
		aSys.PULSE_100MS	:= NOT aSys.PULSE_100MS;
   	aSys.u100ms    	:= 1;
	ELSE
   	aSys.u100ms    := 0;
	END_IF;
	aSys.et200		:= aSys.et200 + SYSTEM_S.LAST_CYCLE_TIME_100US;
	IF aSys.et200 >= 1900 THEN
		aSys.et200			:= 0;
		aSys.PULSE_200MS 	:= NOT aSys.PULSE_200MS;
	END_IF;
	// USINT
	aSys.n1Min     := BOOL_TO_USINT(SYSTEM_S.F_EDGE_1MIN);           // kazdu 1.Min bude = 1
	aSys.n100ms    := BOOL_TO_USINT(SYSTEM_S.F_EDGE_100MS);     //;
	aSys.n50ms     := BOOL_TO_USINT(SYSTEM_S.R_EDGE_100MS OR SYSTEM_S.F_EDGE_100MS);     //;
	// UINT
	aSys.u1Min     := BOOL_TO_UINT(SYSTEM_S.F_EDGE_1MIN);           // kazdu 1.Min bude = 1
  	aSys.i1Min     := USINT_TO_INT(aSys.n1Min);           			// MIN	: INT
	// 1. sec
	IF SYSTEM_S.F_EDGE_1SEC THEN
   	aSys.n1Sec     := 1;           								// SEC	: USINT
  		aSys.u1Sec     := 1;           								// SEC	: UINT
	ELSE
   	aSys.n1Sec     := 0;
  		aSys.u1Sec     := 0;
	END_IF;
	aSys.cyc     		:= NOT aSys.Cyc;							// kazdy cyklus sa prepne
	aSys.RestCyc   	:= aSys.RestCyc + 1;

	CASE aSys.ini OF
       0:	// riadna prevadzka
			// sekvencia 3 cyklov za sebou po prechode na novu minutu, alebo natvrdo zadanim aSys.RefCycNew := true
			// 1 -> 2 -> 3 ->  0
			CASE aSys.RefCyc OF
				0:  IF aSys.RefCycNew THEN										// je zaradena nova poziadavka na restart sekvencie - zacne az ked skonci predchadzajuca sekvencia
						aSys.RefCyc		:=	1;
						aSys.RefCycNew	:= false;
					END_IF;
				3:	// obehlo 3x
					aSys.RefCyc	:=	0;
			ELSE
					aSys.RefCyc := aSys.RefCyc + 1;                 // rucne sa moze nastartovat hocikde v programe na (1), tu sa prida na (2)
			END_CASE;
(*
               Paradox( chan_code := CH5_uni, par_system_data := paradox_data,
                         max_zone_count  := paradox_max_zone_count);
               aSys.ExtPSN := Paradox.com_ok;
*)

(*)
            IF SYSTEM_S.F_EDGE_1DAY OR aSys.Restart THEN                   // novy den
					aSys.RefCyc	:=	1;														// v dalsom cykle nastartuje TypDay
	  				aMeteo.SunriseTime := SunTime( direction := Sunrise, zenith := Zenith_Official,
   		                       longitude := xGlb^.cx.longitude, latitude := xGlb^.cx.latitude,
      		                    utcOffset := UtcOffset_CR(), actDate := aSys.NhDate);
				  	aMeteo.SunsetTime := SunTime( direction := Sunset, zenith := Zenith_Official,
			   		             longitude := xGlb^.cx.longitude, latitude := xGlb^.cx.latitude,
               		          utcOffset := UtcOffset_CR(), actDate := aSys.NhDate);
					xHom^.ok.ref := true;
				ELSIF SYSTEM_S.F_EDGE_1MIN  THEN												// nastartuje 1.cyklus  - ma prednost pred vsetkym
					aSys.RefCyc	:=	1;                                  				// prvy cyklus kde sa skutocne zacne robit ma cislo  2, 3-4-5
					_NhSysUpd(fDbx:=true, file:=1);                                // Mem->RBx, ked bude file > 10 aj RBx->file
				ELSIF aSys.RefCyc	= 0 THEN
					IF aSys.RefCycNew THEN										// je zaradena nova poziadavka na restart sekvencie - zacne az ked skonci predchadzajuca sekvencia
						aSys.RefCyc		:=	1;
						aSys.RefCycNew	:= false;
					END_IF;
				ELSIF aSys.RefCyc	> 3 THEN                         	// pocita 4 cyklov za sebou od prechodu  [2..6]
					aSys.RefCyc	:=	0;
				ELSE
					aSys.RefCyc := aSys.RefCyc + 1;                 // rucne sa moze nastartovat hocikde v programe na (1), tu sa prida na (2)
				END_IF;
*)
            { $ IFDEF __NH_WEB }
               fbWebControl();
            { $ END_IF }                      // zobrazenie nastavenych DEV - za DEV. Ak sa nieco prestavi vo web v dalej otocke sa to prejavi v DEV
            { $ IFDEF __NH_WRK }
               _NhDataWrk();
			{ $ END_IF }

//         _NhDevControl();           // fyzicke nastavenie DEV, malo buy byt prve
			fbNotify();
			fbWebPush();

			aSys.F_EDGE_1MIN		:= FALSE;		// vynuluje sa edge
			aSys.F_EDGE_1HOUR		:= FALSE;		// vynuluje sa edge
			aSys.F_EDGE_1DAY		:= FALSE;		// vynuluje sa edge
			aSys.F_EDGE_1MON		:= FALSE;		// vynuluje sa edge
			aSys.F_EDGE_1YEAR		:= FALSE;		// vynuluje sa edge
			aSys.Restart  			:= false;                     						// vynuluje sa restart, ale az ked sa prebehu prvykrat vsetky DEV

     	10:    ;  // nic
            rb             := _NhSysLogMsg(msg:='Check data: _Nh_DEV_RESTART');
		     	_Nh_DEV_RESTART();
            rb       		:= _NhSysLogMsg(eRowAfter:=1,msg:='*** KONIEC RESTARTU ***');
            _NhCloseAllFiles();
            aSys.ini       := 0;

		11:	// vytvori HET
				fbCrHet();
				IF aSys.ini = 0 THEN
//			      fbCrDir.go		:= -2000;
      		END_IF;

(*
     	49:    // este raz pootvarat vsetky subory
				_NhCloseAllFiles();
//				aSys.OpenFilesCount := OpenFilesCount();
      		aSys.ini    := 10;

*)
(*
            IF fbCrDir.Done THEN
               yTx2     	:= 'UKONCENE vytvaranie LOG adresarov [49]';
               rb       	:= _Nh1RowTxt(logRst:=1);
	            aSys.ini    := 10;
            END_IF;
            fbCrDir();
*)
     	40:    // Upload program

//				yTx2           := CONCAT('start LoadNewPackage2:',yTx4);
            rb             := _Nh1RowTxt(logRst := 1, adTime:=3, EmpRow:=1);
				ok 				:= LoadNewPackage2( rq := true, pckg := yTx4);
            yTx2           := CONCAT('End LoadNewPackage2:',BOOL_TO_STRINGF(ok,'%b{Yes^No}' ));
            rb             := _Nh1RowTxt(logRst := 1, adTime:=3);
				aSys.ini			:= 0;

     	50:    // upravena ram do DBX
            _Nh_Go_MemToDBX();
            yTx2  := 'Na zaver upravena  RAM->DBX';
            rb             := _Nh1RowTxt(logRst := 1);
				aSys.ini       := 10;

		100:	// ulozit RAM do DBX a spustit zalohovanie dobrej DBX na SDC
            _NhWrkRam();                  // adresy WRK ram za poslednymi datami
            aSys.ini       := 50;

   	180:    // export VAZ[1..4]
				cf 		:= 1;
				nd			:= 1;
				_NhxVaz(cv:=cf,nd:=nd);
           	aSys.ini := 181;
   	181:    //
		    	IF _Nh_Vaz_LOG_CV() THEN
					cf 		:= 2;
					nd			:= 1;
					_NhxVaz(cv:=cf,nd:=nd);
	            aSys.ini       := 182;
		    	END_IF;
   	182:    //
		    	IF _Nh_Vaz_LOG_CV() THEN
					cf 		:= 3;
					nd			:= 1;
					_NhxVaz(cv:=cf,nd:=nd);
	            aSys.ini       := 183;
		    	END_IF;
   	183:    //
		    	IF _Nh_Vaz_LOG_CV() THEN
					cf 		:= 4;
					nd			:= 1;
					_NhxVaz(cv:=cf,nd:=nd);
            aSys.ini       := 184;
//	            aSys.ini       := 100;
		    	END_IF;
   	184:    //
	            aSys.ini       := 100;
		    	IF _Nh_Vaz_LOG_CV() THEN
	            aSys.ini       := 100;
		    	END_IF;

		190:    // skontroluje a prida POI
            _Nh_POI_INI();
(*
				IF _GoExp THEN
           		aSys.ini       := 180;
				ELSE
           		aSys.ini       := 100;
				END_IF;
*)

 aSys.ini := 100;

    	200:    // otestuje vazby a ich parametre
            { $IFDEF __NH_WRK }
               _NhDataWrk();
            { $END_IF }
            _NhIniVAZ();
            aSys.ini := 190;

(*
    	210:    // skontroluje konzistenciu ROM,SBJ ....., nastartuje parametre
            _Nh_Ini_DEV_Test();
           	aSys.ini       := 213;
*)

    	213:    // otestuju sa postupne vsetky CFG prida parametre k DEV
            _Nh_Ini_PAR_Test();

    	214:    // koniec testu parametrov
            aSys.ini := 200;

    	217:    // len pre testovanie,
// _NhIsObrOk(frm:=260);

            { $IFDEF __NH_WRK }
               _NhDataWrk();

            { $END_IF }

////***********************

    	220:    // dorobi default vety + CAT,USR,FAV,HET ...,
            _Nh_Ini_DEFAUL_CFG();    							// dorobi default data

//				aSys.ini := 217;
//RETURN;

            aSys.CfgRamOk  := true;
            _Nh_Go_MemToDBX();                           // ulozi aktualnu RAM do DBX
				aSys.ini := 222;

	 	222:    // START Import dev+HW address CIB
				yTx2 		:= 'START Import CIB';
				_Nh1RowTxt(logRst:=1); //,EmpRow:=1);
				fb_Nh_Import_CIB(Go:=1);
            { $IFDEF __NH_WRK }
               _NhDataWrk();
            { $END_IF }
				aSys.Ini 		:= 223;
	 	223:    // Running Import CIB
            fb_Nh_Import_CIB();
				IF fb_Nh_Import_CIB.err THEN
					aSys.Ini 	:= 217;
				ELSIF fb_Nh_Import_CIB.done THEN
					yTx2 	:= 'END Import CIB';
					_Nh1RowTxt(logRst:=1);
					aSys.Ini 	:= 225;
   			END_IF;

    	225:    // skontroluje konzistenciu ROM,SBJ ....., nastartuje parametre

            _Nh_Ini_DEV_Test();
				aSys.exp			:= 0;
           	aSys.ini       := 213;

    	229:    // Err section 22x
				;

(*	RESTART
	250		skontroluje DBx,RBx
				_Nh_CUST_RESTART()
	251		_Nh_Create_DIR(Go:=1)
	240-242	fb_Nh_Create_FRM	COPY NH2/200/FRM/*.* -> RAM/FRM/
	230		zisti ci mame MEM niekde zalohovanu v poradi
				1.RBx .. _NhIsDBxCfgOk(RBx:=true)
				2.File   aSys.CfgBckOk {oznaci_NhIsDBxCfgOk() }
				3.DBx	   _NhIsDBxCfgOk(), ak sa najde prekopiruje sa do RBx: DBx->RBx
	231-232	Load&Convert Old CFG->Mem (z: RBx alebo DBx)
	220		_Nh_Ini_DEFAUL_CFG() - dorobi default data
	222-223	fb_Nh_Import_CIB() :	Import dev+HW address CIB
	225		_Nh_Ini_DEV_Test()	- zakladne testy konzistencie
	213-214 	_Nh_Ini_PAR_Test();	- testy PAR + prida nove PAR
	200		_NhIniVAZ(); 			- konzistenia vazieb
	190		_Nh_POI_INI();      	- skontroluje a prida POI
	100-50	 _Nh_Go_MemToDBX(); 	- 'Na zaver upravena  RAM->DBX';
	10			_Nh_DEV_RESTART(),_NhCloseAllFiles();	- pozatvara vsetky subory na SDC a otvori _NhLangTxt
*)

	 	230:    // find CFG (aMem) in RamBox/DataBox/SDC, then copy to RamBox and then RBx->Mem
			 	IF aSys.NewDBX THEN
					aSys.CfgBckOk	:=	false;
					aSys.UseRBx	   := aSys.IS_RBx;
					rb:=_NhSysLogMsg(msg:='NEW Cfg requested !');
					aSys.Ini			:= 220;
				ELSE
					fb_Nh_Cfg_Backup.IniEnd:=230; fb_Nh_Cfg_Backup.IniErr:=239; fb_Nh_Cfg_Backup.IniRun:=255;	// predbezne
					IF aSys.IS_RBx  THEN																			// from RamBox
						IF _NhIsDBxCfgOk(RBx:=true) THEN                      						// v RBx je obraz mem
    						yTx2  		:= '->RamBOX OK.';
							aSys.UseRBx	:= true;
							aSys.Ini 	:= 231;
						ELSIF aSys.CfgBckOk THEN      															// na zaciatku je 0, potom nastavi
    						yTx2  			:= '...No-RBx,but File.Ok.{File->RBx}';
							fb_Nh_Cfg_Backup.Go		:= 12; 																		// file->RAM, next back here
						ELSIF _NhIsDBxCfgOk(RBx:=false) THEN                      					// v DBX je obraz mem
    						yTx2  		:= '..DBX-Ok.{DBX->File}';
							fb_Nh_Cfg_Backup.Go	:= 3;	   																// DBX->File
						ELSE
   	 					yTx2  			:= '...No RBx/DBx/File -> {Go empty: NewDBX=true}';
							aSys.NewDBX    := true;
						END_IF;
  					ELSIF aSys.CfgBckOk THEN																	// after
  						yTx2  := '...CPU has no RamBox,but File from DBx.Ok.{now File->Mem}';
						fb_Nh_Cfg_Backup.Go:=11; fb_Nh_Cfg_Backup.IniEnd:=220;												// file->Mem
						aSys.UseRBx	:= false;
					ELSIF _NhIsDBxCfgOk(RBx:=false) THEN                      						// v DBX je obraz mem
  						yTx2  		:= '..CPU has no RamBox,but DBX-Ok.{DBX->File}';
						fb_Nh_Cfg_Backup.Go	:= 3;	   																	// DBX->File, next back here
						aSys.UseRBx	:= true;
					ELSE
						yTx2 			:= 'CPU has no RamBox, and NOT DBX. {Go empty: NewDBX=true}';
						aSys.NewDBX := true;
					END_IF;
					rb:=_NhSysLogMsg(msg:=yTx2);
				END_IF;
//				aSys.Ini := 226;

	 	231:    // START 1.Import CFG DBX->Mem
				yTx2 		:= CONCAT('START Load & Convert Old CFG: ',BOOL_TO_STRINGF(aSys.UseRBx,'%b{Rbx^DBX}'),'->Mem.',BOOL_TO_STRINGF(xDbx^.FromDBx128,' DBx128: %b{Y^N}') );
				_Nh1RowTxt(logRst:=1); //,EmpRow:=1);
	         fb_Nh_Cfg_Restart(init:=1, wh:=0, cx:=1);
				aSys.Ini 		:= 232;

	 	232:    // Running Load Old CFG
            fb_Nh_Cfg_Restart();
				IF fb_Nh_Cfg_Restart.done THEN
					yTx2 	:= 'END Load Old CFG';
					_Nh1RowTxt(logRst:=1);
					aSys.Ini 	:= 220;
   			END_IF;

		238:    ;	//Error section 230
		239:    ;	//Error section 230
				;

	 	240:    // aktualne formulare -> NH2/200/FRM
            { $ IFDEF __NH_FRM }
					IF fb_Nh_Create_FRM.done THEN
						yTx2 		:= 'OK. New FRM';
  		 				rb 		:= _Nh1RowTxt(logRst := 1);
		            aSys.ini := 241;
					ELSIF fb_Nh_Create_FRM.busy THEN ;
					ELSE 	fb_Nh_Create_FRM(Go:=1,all:=true);
					END_IF;
					fb_Nh_Create_FRM();
            { $ ELSE }
					aSys.ini := 241;
            { $ END_IF }

		241:   // COPY NH2/200/FRM/*.* -> RAM/FRM/
         	IF aSys.DiskHed.Disk[4].Exist THEN												// RAM exist, go copy
   				_Nh_Log_Path(wh:=24, frm:=1, wh2:=1);                                  // yTx3,yTx4
	     			yTx2 		:= CONCAT('START Copy {',yTx3,'}->{',yTx4,'}');													// START Create Dir
              	rb      	:= _Nh1RowTxt(logRst := 1);
              	fb_Nh_Copy_Dir(init:=TRUE,Go:= 2,IniRun:=255,IniEnd:=242,IniErr:=249);
            ELSE
              	aSys.Ini := 230;
            END_IF;
	 	242:    // End Copy
				yTx2		:= CONCAT('END   Copy  f: ',UINT_TO_STRING(fb_Nh_Copy_Dir.files),' s: ',UDINT_TO_STRING(fb_Nh_Copy_Dir.allSize) )  ;
    			rb			:= _Nh1RowTxt(logRst := 1);
      		aSys.Ini := 230;
	 	249: 	// Err Copy Dir
				;
	 	250: 	// restart
  				//          aSys.prgChange    		:= PROGRAMISCHANGED();
				rb:=_NhCloseAllFiles();
				IF CPU_CODE >= 2000 THEN
					rb 					:= ResizeRamBox( newSize := 16*1024);   	// 16MB*1024 = 16384 kByte
					aSys.Size_RBx 		:= UINT_TO_UDINT( SizeOfRamBox() ) * 1024;   							// 128 kb   (128*1024=131072 Byte)
					aSys.IS_RBx			:= aSys.Size_RBx >= 16777216;
				ELSE
					aSys.IS_RBx			:= false;
					aSys.Size_RBx 		:= 0;
//					yTx1					:= 'WWW/LOGS/';
			  	END_IF;
				yTx1						:= 'WWW/NH2/';
				rb							:=	DirCreate( dirName := yTx1 );																	// create default LOG adr
				aSys.Restart     		:= TRUE;
				aSys.RefCyc				:=	1;
//				aSys.rst.In				:= true;
				aSys.CfgBckOk			:=	FALSE;																	// flag, that BckFile no-Exiat
				aSys.Size_DBx 			:= UINT_TO_UDINT( SizeOfDataBox()) * 1024;   								// 128 kb   (128*1024=131072 Byte)
				aSys.IS_DBX				:= aSys.Size_DBx >= 131072;

//				aSys.DiskHed.USB_Ready.In	:= SYSTEM_S.USB_DISK_READY;									// vynuluje sa flag USB ready
//				aSys.DiskHed.USB_Ready.Q	:= SYSTEM_S.USB_DISK_READY;									// vynuluje sa flag USB ready

				aDbx.aCfx[0]   := _cfg0;
		   	aDbx.aCfx[1]   := _par0;
	   		aDbx.aCfx[2]   := _vaz0;
		   	aDbx.vRam   	:= _Ram0;                                                         // volna ram
	      	_NheRAM();                                                                    // vymaze virtualnu RAM od vRam (za CFG/PAR/VAZ...
		   	FOR i := 2  TO _Nh_Cfg DO                                                     // offset default Empty vety
    				aCfg[i].ofs   := aCfg[i-1].ofs + aCfg[i-1].siz;
	   		END_FOR;
     			FOR i := 2  TO _Nh_Par DO                                                     // offset default Empty vety
     				aPar[i].ofs   := aPar[i-1].ofs + aPar[i-1].siz ;
     			END_FOR;
				RandomU(seed := _NhSeed, init:=true);

//				rb	:= SetValueToRamBox(ramBoxAddress:=0, length:=_NH_RAM, value := 0);

//				_Nh_CUST_RESTART();                          											// nejake vlasne veci po restarte

				IF IS_COLD_RESTART_PLC 		THEN	yTx0:='COLD';
				ELSIF IS_HOT_RESTART_PLC   THEN  yTx0:='HOT';
				ELSIF IS_RESTART_PLC       THEN  yTx0:='RST';
				ELSE 						      	   yTx0:='UNKNOWN';
				END_IF;

				SYSTEM_S.F_EDGE_1DAY 	:= true;												// simulate new day for refresh day in room/het
            aSys.Ini 					:= 251;

    	251: 	// 2.cyc After restart - create dir OK

				rb:=_NhSysLogMsg(write:=1,eRowBefore:=1,msg:=' *** '+yTx0+' RESTART ***   DBx: '+UINT_TO_STRING(SizeOfDataBox())+' kB, RBx: '+UINT_TO_STRING( SizeOfRamBox() )+BOOL_TO_STRINGF(SYSTEM_S.USB_DISK_READY, ' kB; USB:%b{Y^N}')+'   *** ');				rb:=_NhSysLogMsg(eRowAfter:=1,NoTime:=1,msg:=DT_TO_STRINGF(_NhLastPowerOffState.LastDt, '%TYY.MM.DD-hh:mm:ss.zzz ') +',Ini:='+USINT_TO_STRING(_NhLastPowerOffState.ini) );
//				_Nh_Log_Dbx_ADD(ev:='AL1',src:='PIR',key:='Pir-1',val:='On',subj:=1,rom:=101);
            aSys.Ini 				:= 241;

//            aSys.Ini 				:= 255;

	 	252:    // test
            ;
		254:    // Error
            ;
		255:    // running more like one cycle, block all function except fb_ ....
            ;
	END_CASE;

	// time events - change progtam date
	IF SYSTEM_S.F_EDGE_1DAY  THEN				   											// novy den
		aSys.F_EDGE_1DAY	:= true;														// NH event
		aSys.F_EDGE_1MON 	:= aSys.MONTH 	<> SYSTEM_S.COUNTER_MONTHS;												// NH event
		aSys.F_EDGE_1YEAR	:= aSys.YEAR 	<> SYSTEM_S.COUNTER_YEARS;
		aSys.YEAR 			:= SYSTEM_S.COUNTER_YEARS;								// Nh month
		aSys.MONTH 			:= SYSTEM_S.COUNTER_MONTHS;							//	Nh month
		aSys.DAY				:= SYSTEM_S.COUNTER_DAYS_OF_MONTH;					// Nh month
		aSys.RefCycNew		:= true;														// v dalsom cykle nastartuje TypDay
		aSys.YYYY_MM		:= CONCAT(USINT_TO_STRINGF(aSys.YEAR, '20%02d'),'_',USINT_TO_STRINGF(aSys.MONTH, '%02d'),'/');
		fb_Nh_Create_DIR.exec	:= aSys.F_EDGE_1MON ;							// vytvori nove adresare pre novy mesiac
	ELSIF  SYSTEM_S.F_EDGE_1MIN  THEN                   									// new min
		aSys.F_EDGE_1MIN			:= true;												// NH event
		aSys.F_EDGE_1HOUR			:= SYSTEM_S.F_EDGE_1MIN;						// NH event
		aSys.RefCycNew				:= true;												// v dalsom cykle nastartuje TypDay
		// after xxx seconds of error-free operation, make a CFG backup
	ELSIF  SYSTEM_S.F_EDGE_10SEC  THEN                   									// new min
		_NhSysUpd(file:=255);															// Mem->RBx, ked bude file > 10 aj RBx->file
	ELSIF aSys.RestartBck = false THEN										// este nebol urobeny backup po restarte
		IF  aSys.ini = 0 AND SYSTEM_S.COUNTER_1SEC > 4 THEN     						// 1min after restart, create backup file
			IF _NhSysUpd(file:=255) THEN												// Mem->RBx, ked bude file > 10 aj RBx->file
				aSys.RestartBck 	:= true;
			END_IF;
		END_IF
	END_IF;

//	fb_RbxToFile(fileName:=yTx1); //,exec:=FALSE);				// write RamBox -> file
//	- 	exec	0->1; busy:=1; done:=0;	err:=0; 	errID=0;		Open file
//	- 	exec		1  busy:=0; done:=X;	err:=Y; 	errID=Y;		when done or err, will remain X or Y
//	- 	exec	1->0  busy:=0; done:=0;	err:=0; 	errID=0;		reset all
//	- 	err	0->1;	busy:=0;	done:=0;	err:=1;	errID>0;		close file
//	- 	done	0->1;	busy:=0;	done:=1;	err:=0;	errID=0;		close file

//	fb_RbxFromFile(fileName:=yTx1);				// read  file -> RamBox
//	fb_Nh_ToFromFile();

	fb_Nh_Create_DIR();												// test and create directories
	fb_Nh_Cfg_Backup();      	// save from mRam[] to file, or restore to mRam[] from file
	fb_Nh_Copy_Dir();

//	fb_Nh_Log_DBX_RW();		// write log to buffer (DBx,RBx) and read from buffer and send datagram to Pi or Write to USB/LOG
//	fb_Nh_PLC_DIR();

	_NhLastPowerOffState.LastDt	:= aSys.NhDT;
	_NhLastPowerOffState.ini 	:= aSys.ini;
//	_NhLastStateON.ini 		:= aSys.ini;

END_PROGRAM
